FUNCTION F_ScrollListY (* Compute Container_Scrolling_Content.Top (s16Yposition for Q_ChildPosition) from the current row position: -(i32Pos * i32RowHeight). *)
  (* Standard: 61499-2; Description: Copyright (c) 2026 Meisterschulen am Ostbahnhof This program and the accompanying materials are made available under the terms of the Eclipse Public License 2.0 which is available at https://www.eclipse.org/legal/epl-2.0/ SPDX-License-Identifier: EPL-2.0 *)
  (* Version 1.0, 2026-08-09, Franz Höpfinger, Meisterschulen am Ostbahnhof, initial API and implementation and/or initial documentation *)
  PACKAGE isobus::UT::Q::helpers;
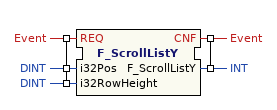
  EVENT_INPUT
    REQ WITH i32Pos, i32RowHeight;
  END_EVENT
  EVENT_OUTPUT
    CNF WITH F_ScrollListY;
  END_EVENT
  VAR_INPUT
    i32Pos : DINT;
    i32RowHeight : DINT;
  END_VAR
  VAR_OUTPUT
    F_ScrollListY : INT;
  END_VAR
  BODY IN ST:
PACKAGE isobus::UT::Q::helpers;

(* Compute Container_Scrolling_Content.Top (s16Yposition for Q_ChildPosition) from the current
 * row position: -(i32Pos * i32RowHeight). *)
FUNCTION F_ScrollListY : INT

VAR_INPUT
	i32Pos : DINT;
	i32RowHeight : DINT;
END_VAR

F_ScrollListY := DINT_TO_INT(-(i32Pos * i32RowHeight));

END_FUNCTION
  END_BODY
END_FUNCTION
